FUNCTION_BLOCK S7_WRITE
  {SET_ATTRIBUTE(OpcUa, SERVICE)}
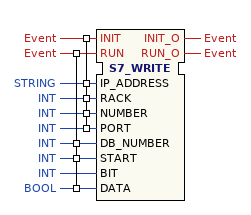
  EVENT_INPUT
    INIT WITH IP_ADDRESS, RACK, NUMBER, PORT;
    RUN WITH DB_NUMBER, START, SIZE, DATA;
  END_EVENT
  EVENT_OUTPUT
    INIT_O;
    RUN_O;
  END_EVENT
  VAR_INPUT
    IP_ADDRESS : STRING; {SET_ATTRIBUTE(OpcUa, Constant.RUN)}
    RACK : INT; {SET_ATTRIBUTE(OpcUa, Constant.RUN)}
    NUMBER : INT; {SET_ATTRIBUTE(OpcUa, Constant.RUN)}
    PORT : INT; {SET_ATTRIBUTE(OpcUa, Constant.RUN)}
    DB_NUMBER : INT; {SET_ATTRIBUTE(OpcUa, Variable.RUN)}
    START : INT; {SET_ATTRIBUTE(OpcUa, Variable.RUN)}
    BIT : INT; {SET_ATTRIBUTE(OpcUa, Variable.RUN)}
    DATA : BOOL; {SET_ATTRIBUTE(OpcUa, Variable.RUN)}
  END_VAR
END_FUNCTION_BLOCK
